PROGRAM P_Patlite
VAR
	bRedLed				AT %Q* :BOOL;				//パトライト赤LED ターミナル5(EL2088)チャンネル5
	bGreenLed			AT %Q* :BOOL;				//パトライト緑LED ターミナル5(EL2088)チャンネル6
	bBlueLed			AT %Q* :BOOL;				//パトライト青LED ターミナル5(EL2088)チャンネル7
	bBuzzerON			AT %Q* :BOOL;				//パトライトブザー ターミナル5(EL2088)チャンネル8
	
	bSwitch				AT %I* :BOOL; 				//パトライトスイッチ ターミナル5(EL1088)チャンネル8

	eLedColor			:E_LedColor;
	fbREdge				:R_TRIG;
	bBuzzerFlag			:BOOL;
	tBlinkTime			:TIME;
	fbTonBlink1			:ton;
	fbTonBlink2			:ton;
END_VAR

//---マシーンステートごとにパトライトを制御---
CASE GVL.eMachineState OF
	
E_MachineState.Emergency:
	eLedColor:=E_LedColor.Red;
	tBlinkTime:=T#100MS;
	IF bBuzzerFlag=FALSE THEN
		bBuzzerON:=TRUE;
	END_IF

E_MachineState.Warning:
	eLedColor:=E_LedColor.Red;
	tBlinkTime:=T#100MS;
	IF bBuzzerFlag=FALSE THEN
		bBuzzerON:=TRUE;
	END_IF

E_MachineState.Stop:
	eLedColor:=E_LedColor.Yellow;
	tBlinkTime:=T#0S;
	bBuzzerON:=FALSE;
	bBuzzerFlag:=FALSE;
	
E_MachineState.Stay:
	eLedColor:=E_LedColor.White;
	tBlinkTime:=T#0S;
	bBuzzerON:=FALSE;
	bBuzzerFlag:=FALSE;
	
E_MachineState.Moving:
	eLedColor:=E_LedColor.Green;
	tBlinkTime:=T#0S;
	bBuzzerON:=FALSE;
	bBuzzerFlag:=FALSE;
	
END_CASE;

//---スイッチが押されたらブザー停止---
IF bSwitch=TRUE THEN
	bBuzzerON:=FALSE;
	bBuzzerFlag:=TRUE;
END_IF

//---ブリンク用のタイマー---
fbTonBlink1(IN:=NOT fbTonBlink2.Q,PT:=tBlinkTime,Q=>fbTonBlink2.IN,ET=>);
fbTonBlink2(IN:=,PT:=tBlinkTime,Q=>,ET=>);


//---LEDを点灯制御---
IF fbTonBlink1.Q=FALSE OR tBlinkTime=T#0S  THEN;
	CASE eLedColor OF
	E_LedColor.Red:
		bRedLed:=TRUE;
		bGreenLed:=FALSE;
		bBlueLed:=FALSE;
	
	E_LedColor.Green:
		bRedLed:=FALSE;
		bGreenLed:=TRUE;
		bBlueLed:=FALSE;	
	
	E_LedColor.Blue:
		bRedLed:=FALSE;
		bGreenLed:=FALSE;
		bBlueLed:=TRUE;
		
	E_LedColor.Yellow:
		bRedLed:=TRUE;
		bGreenLed:=TRUE;
		bBlueLed:=FALSE;
	
	E_LedColor.Cyan:
		bRedLed:=FALSE;
		bGreenLed:=TRUE;
		bBlueLed:=TRUE;
	
	E_LedColor.Purple:
		bRedLed:=TRUE;
		bGreenLed:=FALSE;
		bBlueLed:=TRUE;
	
	E_LedColor.White:
		bRedLed:=TRUE;
		bGreenLed:=TRUE;
		bBlueLed:=TRUE;
	
	E_LedColor.Black:
		bRedLed:=FALSE;
		bGreenLed:=FALSE;
		bBlueLed:=FALSE;
	END_CASE
ELSE;
	bRedLed:=FALSE;
	bGreenLed:=FALSE;
	bBlueLed:=FALSE;
END_IF;

END_PROGRAM

(* stored: Version 1.1.0.1, ProductVersion 3.1.4024.12
   POU P_Patlite: Id {a5bb9a40-855c-4dd1-9843-b749d06b4679}, SpecialFunc None *)
